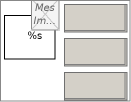
VISUALIZATION VISU_VANNE_3P_H  // 131x102
VAR_IN_OUT
	m_Input_Vanne	:	BLOCK_VVAT_3P;
END_VAR
    Rectangle (4,15 51x44), invisible if: TRUE
    Polygon (0,0), colour toggle: m_Input_Vanne.STATE_Lam
    Rectangle (13,25 44x21), "%s", text variable: m_Input_Vanne.MNEMO
    Polygon (0,0), colour toggle: m_Input_Vanne.STATE_On, invisible if: NOT (m_Input_Vanne.STATE_Off or m_Input_Vanne.STATE_On)
    Button (64,4 63x28), input disabled if: NOT m_Input_Vanne.AUTOR_On_IHM OR NOT .PRG_USER.ACTU_USER.MAINTENANCE, text list: 'TextList_VVAT_3P', text index: 0
        OnMouseClick: toggle m_Input_Vanne.M_On
    Button (64,38 63x28), input disabled if: NOT m_Input_Vanne.AUTOR_Lam_IHM OR NOT .PRG_USER.ACTU_USER.MAINTENANCE, text list: 'TextList_VVAT_3P', text index: 2
        OnMouseClick: toggle m_Input_Vanne.M_Lam
    Button (64,72 63x28), input disabled if: NOT m_Input_Vanne.AUTOR_Off_IHM OR NOT .PRG_USER.ACTU_USER.MAINTENANCE, text list: 'TextList_VVAT_3P', text index: 1
        OnMouseClick: toggle m_Input_Vanne.M_Off
    Image (31,-2 28x32), invisible if: NOT m_Input_Vanne.STATE_Nok, image: MesImages.warning
END_VISUALIZATION

(* stored: Version 1.1.0.1, ProductVersion 3.1.4026.18
   Visu VISU_VANNE_3P_H: Id {48af5ff3-e772-4349-8b63-889cd3ea5fbc} *)
